Universal Robots PolyScope program: d_a.urp

Program d_a (installation=string_planes directory=/programs createdIn=5.17.3 lastSavedIn=5.17.3 robotSerialNumber=20245501435)
Calibrated DH parameters: a=[0.000154, -0.137004, -0.385524, -0.00002, 0.000092, 0]; d=[0.162441, 211.794786, -230.585024, 18.923638, 0.099786, 0.09951]; alpha=[1.569493, -0.001902, 0.003874, 1.570111, -1.570167, 0]; deltaTheta=[0, -1.242934, 1.056292, 0.186646, 0.000002, 0.000001]
InitVariablesNode
Robot Program (runOnlyOnce=true)
  MoveJ speed 60 deg/s, acceleration 80 deg/s^2 (useActiveTCP=true) feature=Base
    Waypoint Waypoint_5 (Relative): relativeFromPosition TCP in base x=331.965 y=722.317 z=108.299 mm, rx=-1.645 ry=-2.1081 rz=1.059 rad; joints [-129.708, -21.47, 51.982, -76.269, -76.861, -148.975] deg; TCP offset x=28.21 y=-96.107 z=-99.69 mm, rx=0 ry=0 rz=0 rad; TCP in base x=324.767 y=765.314 z=130.378 mm, rx=-1.4944 ry=-2.2778 rz=1.1569 rad; joints [-127.057, -14.742, 33.543, -62.028, -82.971, -153.445] deg
